FUNCTION_BLOCK IED87 (* Composite Function Block Type *)
  (* Standard: 61499-2 *)
  (* Version 1.0, 2021-03-01, badger *)
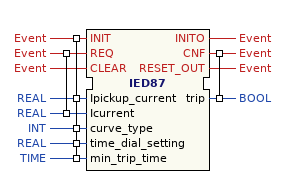
  EVENT_INPUT
    INIT WITH Ipickup_current, min_trip_time, time_dial_setting, curve_type; (* Initialization Request *)
    REQ WITH Icurrent; (* Normal Execution Request *)
    CLEAR;
  END_EVENT
  EVENT_OUTPUT
    INITO; (* Initialization Confirm *)
    CNF WITH trip; (* Execution Confirmation *)
    RESET_OUT;
  END_EVENT
  VAR_INPUT
    Ipickup_current : REAL; (* in amps *)
    Icurrent : REAL; (* in amps *)
    curve_type : INT; (* one of the ANSI_Time_Curves enumerated types *)
    time_dial_setting : REAL; (* typically 0.5 to 15 *)
    min_trip_time : TIME; (* in milliseconds *)
  END_VAR
  VAR_OUTPUT
    trip : BOOL; (* Output event qualifier *)
  END_VAR
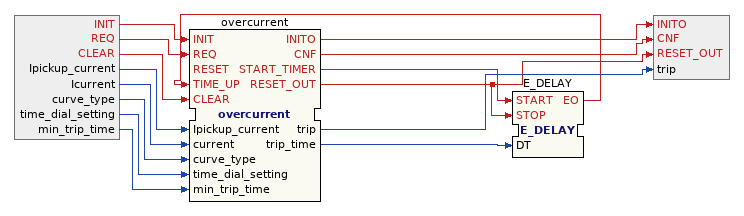
  FBS
    overcurrent : overcurrent;
    E_DELAY : E_DELAY;
  END_FBS
  EVENT_CONNECTIONS
    INIT TO overcurrent.INIT;
    REQ TO overcurrent.REQ;
    CLEAR TO overcurrent.CLEAR;
    overcurrent.START_TIMER TO E_DELAY.START;
    overcurrent.RESET_OUT TO E_DELAY.STOP;
    overcurrent.INITO TO INITO;
    overcurrent.CNF TO CNF;
    overcurrent.RESET_OUT TO RESET_OUT;
    E_DELAY.EO TO overcurrent.TIME_UP;
  END_CONNECTIONS
  DATA_CONNECTIONS
    Ipickup_current TO overcurrent.Ipickup_current;
    Icurrent TO overcurrent.current;
    curve_type TO overcurrent.curve_type;
    time_dial_setting TO overcurrent.time_dial_setting;
    min_trip_time TO overcurrent.min_trip_time;
    overcurrent.trip_time TO E_DELAY.DT;
    overcurrent.trip TO trip;
  END_CONNECTIONS
END_FUNCTION_BLOCK
